Universal Robots PolyScope program: shaft_v1.urp

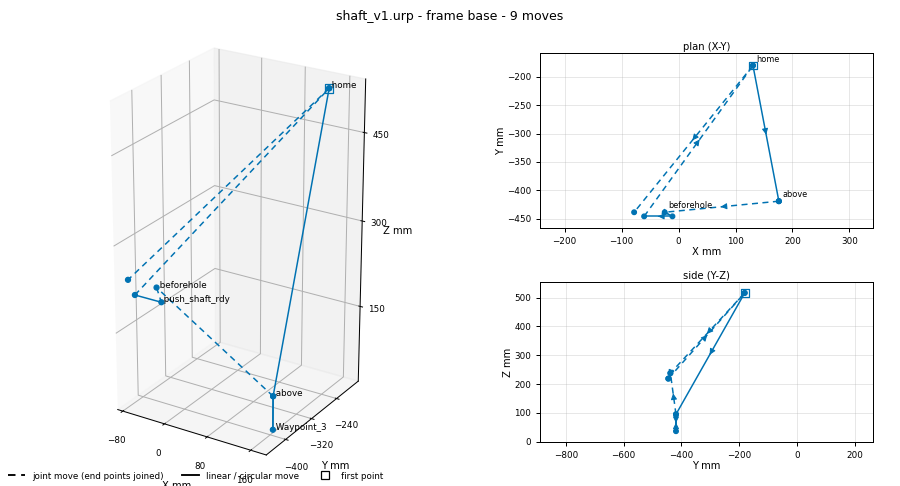
[picture p0: tool path of shaft_v1.urp in frame base, 9 of 9 moves have a stored position in this frame; points joined in program order, loops and branches not executed]
Program shaft_v1 (installation=default directory=/programs/wrs2020 createdIn=5.7.0.90932 lastSavedIn=5.7.0.90932 robotSerialNumber=20205500607)
Calibrated DH parameters: a=[0.000096, -0.337, -0.383372, 0.000118, 0.000015, 0]; d=[0.162724, 79.377998, -95.545185, 16.300583, 0.099689, 0.099499]; alpha=[1.569249, 0.003272, 0.005201, 1.570041, -1.570219, 0]; deltaTheta=[0, 0.65664, 5.410619, 0.215927, -0.000001, 0]
Robot Program (runOnlyOnce=true)
  MoveJ speed 180 deg/s, acceleration 80 deg/s^2 (useActiveTCP=true) feature=Base
    Waypoint home: TCP in base x=130.635 y=-180.692 z=515.97 mm, rx=-0.0117 ry=-3.1402 rz=-0.0315 rad; joints [89.951, -120.324, 80.212, -48.705, -89.957, -0.002] deg; TCP offset x=0 y=0 z=165 mm, rx=0 ry=0 rz=0 rad
  URCap Gripper (Robotiq_Grippers, Robotiq Inc.) dataModel(position=40.0, force=100.0, speed=100.0, positionInDouble=40.0, forceInDouble=100.0, speedInDouble=100.0, slaveIds=[9], blocking=true)
  MoveL speed 250 mm/s, acceleration 1200 mm/s^2 (useActiveTCP=true) feature=Base
    Waypoint above: TCP in base x=176.103 y=-418.817 z=95.382 mm, rx=2.2322 ry=2.1885 rz=0.0336 rad; joints [94.991, -88.211, 123.574, -125.231, -88.184, 96.136] deg
    Waypoint Waypoint_3: TCP in base x=176.103 y=-418.817 z=36.839 mm, rx=2.2322 ry=2.1885 rz=0.0336 rad; joints [94.966, -81.879, 127.739, -135.729, -88.195, 96.172] deg
  URCap Gripper (Robotiq_Grippers, Robotiq Inc.) dataModel(position=100.0, force=100.0, speed=100.0, positionInDouble=100.0, forceInDouble=100.0, speedInDouble=100.0, slaveIds=[9], blocking=true)
  MoveL speed 250 mm/s, acceleration 1200 mm/s^2 (useActiveTCP=true) feature=Base
    Waypoint above: TCP in base x=176.103 y=-418.817 z=95.382 mm, rx=2.2322 ry=2.1885 rz=0.0336 rad; joints [94.991, -88.211, 123.574, -125.231, -88.184, 96.136] deg
  MoveJ speed 60 deg/s, acceleration 80 deg/s^2 (useActiveTCP=true) feature=Base
    Waypoint beforehole: TCP in base x=-24.236 y=-438.216 z=237.961 mm, rx=2.1821 ry=2.2311 rz=0.0137 rad; joints [68.566, -99.136, 110.829, -101.657, -88.409, 67.166] deg
  MoveL speed 20 mm/s, acceleration 500 mm/s^2 (useActiveTCP=true) feature=Base
    SuppressedNode
      Waypoint athole: TCP in base x=-43.043 y=-438.482 z=237.002 mm, rx=2.1821 ry=2.2311 rz=0.0137 rad; joints [66.199, -98.823, 110.698, -101.787, -88.409, 64.799] deg
    MoveDirectionNode (selectedDirection=YMinus) feature=Joint_6_name
      Until TOOL_CONTACT_DETECTION (allowActions=false retraction=0 decelerationAcceleration=3 decelerationAngularAcceleration=34.906585)
  MoveL speed 250 mm/s, acceleration 1200 mm/s^2 (useActiveTCP=true) feature=Base
    MoveDirectionNode (selectedDirection=ZPlus)
      Until DISTANCE (allowActions=false deceleration=3 distanceNodeType=STOP) Distance=0.002; motionParameters(blendRadius=0)
  Force Frame feature=Joint_6_name; selection=[0, 1, 0, 0, 0, 0]; wrench=[-20, -20, 0, 0, 0, 0]; limitsForce=[0.01, 0.01, 0.005, 1.047198, 1.047198, 1.047198]; limitsMotion=[0.1, 0.1, 0.1, 0.349066, 0.349066, 0.349066]
    Wait Sleep waitTime=3
    SuppressedNode
      Loop Counting (count=10) loopVariable(name=Loop_2)
        Force Frame feature=Base; selection=[1, 0, 1, 0, 0, 0]; wrench=[-10, 5, 5, 0, 0, 0]; limitsForce=[0.01, 0.01, 0.01, 1.047198, 1.047198, 1.047198]; limitsMotion=[0.1, 0.1, 0.1, 0.349066, 0.349066, 0.349066]
          Wait Sleep waitTime=2
        Force Frame feature=Base; selection=[1, 0, 1, 0, 0, 0]; wrench=[-10, 5, -5, 0, 0, 0]; limitsForce=[0.01, 0.01, 0.01, 1.047198, 1.047198, 1.047198]; limitsMotion=[0.1, 0.1, 0.1, 0.349066, 0.349066, 0.349066]
          Wait Sleep waitTime=2
        Force Frame feature=Base; selection=[1, 1, 0, 0, 0, 0]; wrench=[-10, 5, 5, 0, 0, 0]; limitsForce=[0.01, 0.01, 0.01, 1.047198, 1.047198, 1.047198]; limitsMotion=[0.1, 0.1, 0.1, 0.349066, 0.349066, 0.349066]
          Wait Sleep waitTime=2
        Force Frame feature=Base; selection=[1, 1, 0, 0, 0, 0]; wrench=[-10, -5, 5, 0, 0, 0]; limitsForce=[0.01, 0.01, 0.01, 1.047198, 1.047198, 1.047198]; limitsMotion=[0.1, 0.1, 0.1, 0.349066, 0.349066, 0.349066]
          Wait Sleep waitTime=2
    'spiral motion'
    SuppressedNode
      Loop Counting (count=30) loopVariable(name=Loop_1)
        MoveL speed 250 mm/s, acceleration 1200 mm/s^2 (useActiveTCP=true) feature=Base
          MoveDirectionNode (toolParams=0.005, 0.02) expression=[sin((Loop_1-1)/6*3.141),0.0,-cos((Loop_1-1)/6*3.141)]; feature=Joint_6_name
            Until DISTANCE (allowActions=false deceleration=3 distanceNodeType=STOP) Distance=0.001; motionParameters(blendRadius=0)
    'grid motion'
    var_1 := 1
    Loop While (checkContinuously=true) expression=( pose_dist(get_actual_tcp_pose(), fully_inserted) > 0.005) and  (var_1 < 6)
      MoveL speed 250 mm/s, acceleration 1200 mm/s^2 (useActiveTCP=true) feature=Base
        MoveDirectionNode (selectedDirection=XPlus toolParams=0.005, 0.02) feature=Joint_6_name
          Until DISTANCE (allowActions=false deceleration=3 distanceNodeType=STOP) Distance=0.0005; motionParameters(blendRadius=0)
        MoveDirectionNode (selectedDirection=ZMinus toolParams=0.005, 0.02) feature=Joint_6_name
          Until DISTANCE (allowActions=false deceleration=3 distanceNodeType=STOP) Distance=0.0005; motionParameters(blendRadius=0)
        MoveDirectionNode (selectedDirection=XMinus toolParams=0.005, 0.02) feature=Joint_6_name
          Until DISTANCE (allowActions=false deceleration=3 distanceNodeType=STOP) Distance=0.0005; motionParameters(blendRadius=0)
        MoveDirectionNode (selectedDirection=XMinus toolParams=0.005, 0.02) feature=Joint_6_name
          Until DISTANCE (allowActions=false deceleration=3 distanceNodeType=STOP) Distance=0.0005; motionParameters(blendRadius=0)
        MoveDirectionNode (selectedDirection=ZPlus toolParams=0.005, 0.02) feature=Joint_6_name
          Until DISTANCE (allowActions=false deceleration=3 distanceNodeType=STOP) Distance=0.0005; motionParameters(blendRadius=0)
        MoveDirectionNode (selectedDirection=XPlus toolParams=0.005, 0.02) feature=Joint_6_name
          Until DISTANCE (allowActions=false deceleration=3 distanceNodeType=STOP) Distance=0.0005; motionParameters(blendRadius=0)
        MoveDirectionNode (selectedDirection=XPlus toolParams=0.005, 0.02) feature=Joint_6_name
          Until DISTANCE (allowActions=false deceleration=3 distanceNodeType=STOP) Distance=0.0005; motionParameters(blendRadius=0)
        MoveDirectionNode (selectedDirection=ZPlus toolParams=0.005, 0.02) feature=Joint_6_name
          Until DISTANCE (allowActions=false deceleration=3 distanceNodeType=STOP) Distance=0.0005; motionParameters(blendRadius=0)
        MoveDirectionNode (selectedDirection=XMinus toolParams=0.005, 0.02) feature=Joint_6_name
          Until DISTANCE (allowActions=false deceleration=3 distanceNodeType=STOP) Distance=0.0005; motionParameters(blendRadius=0)
        MoveDirectionNode (selectedDirection=XMinus toolParams=0.005, 0.02) feature=Joint_6_name
          Until DISTANCE (allowActions=false deceleration=3 distanceNodeType=STOP) Distance=0.0005; motionParameters(blendRadius=0)
        MoveDirectionNode (selectedDirection=ZMinus toolParams=0.005, 0.02) feature=Joint_6_name
          Until DISTANCE (allowActions=false deceleration=3 distanceNodeType=STOP) Distance=0.0005; motionParameters(blendRadius=0)
        MoveDirectionNode (selectedDirection=XPlus toolParams=0.005, 0.02) feature=Joint_6_name
          Until DISTANCE (allowActions=false deceleration=3 distanceNodeType=STOP) Distance=0.0005; motionParameters(blendRadius=0)
      MoveL speed 250 mm/s, acceleration 1200 mm/s^2 (useActiveTCP=true) feature=Base
        MoveDirectionNode (selectedDirection=XPlus toolParams=0.005, 0.02) feature=Joint_6_name
          Until DISTANCE (allowActions=false deceleration=3 distanceNodeType=STOP) Distance=0.001; motionParameters(blendRadius=0)
        MoveDirectionNode (selectedDirection=ZMinus toolParams=0.005, 0.02) feature=Joint_6_name
          Until DISTANCE (allowActions=false deceleration=3 distanceNodeType=STOP) Distance=0.001; motionParameters(blendRadius=0)
        MoveDirectionNode (selectedDirection=XMinus toolParams=0.005, 0.02) feature=Joint_6_name
          Until DISTANCE (allowActions=false deceleration=3 distanceNodeType=STOP) Distance=0.001; motionParameters(blendRadius=0)
        MoveDirectionNode (selectedDirection=XMinus toolParams=0.005, 0.02) feature=Joint_6_name
          Until DISTANCE (allowActions=false deceleration=3 distanceNodeType=STOP) Distance=0.001; motionParameters(blendRadius=0)
        MoveDirectionNode (selectedDirection=ZPlus toolParams=0.005, 0.02) feature=Joint_6_name
          Until DISTANCE (allowActions=false deceleration=3 distanceNodeType=STOP) Distance=0.001; motionParameters(blendRadius=0)
        MoveDirectionNode (selectedDirection=XPlus toolParams=0.005, 0.02) feature=Joint_6_name
          Until DISTANCE (allowActions=false deceleration=3 distanceNodeType=STOP) Distance=0.001; motionParameters(blendRadius=0)
        MoveDirectionNode (selectedDirection=XPlus toolParams=0.005, 0.02) feature=Joint_6_name
          Until DISTANCE (allowActions=false deceleration=3 distanceNodeType=STOP) Distance=0.001; motionParameters(blendRadius=0)
        MoveDirectionNode (selectedDirection=ZPlus toolParams=0.005, 0.02) feature=Joint_6_name
          Until DISTANCE (allowActions=false deceleration=3 distanceNodeType=STOP) Distance=0.001; motionParameters(blendRadius=0)
        MoveDirectionNode (selectedDirection=XMinus toolParams=0.005, 0.02) feature=Joint_6_name
          Until DISTANCE (allowActions=false deceleration=3 distanceNodeType=STOP) Distance=0.001; motionParameters(blendRadius=0)
        MoveDirectionNode (selectedDirection=XMinus toolParams=0.005, 0.02) feature=Joint_6_name
          Until DISTANCE (allowActions=false deceleration=3 distanceNodeType=STOP) Distance=0.001; motionParameters(blendRadius=0)
        MoveDirectionNode (selectedDirection=ZMinus toolParams=0.005, 0.02) feature=Joint_6_name
          Until DISTANCE (allowActions=false deceleration=3 distanceNodeType=STOP) Distance=0.001; motionParameters(blendRadius=0)
        MoveDirectionNode (selectedDirection=XPlus toolParams=0.005, 0.02) feature=Joint_6_name
          Until DISTANCE (allowActions=false deceleration=3 distanceNodeType=STOP) Distance=0.001; motionParameters(blendRadius=0)
      var_1 := var_1+1
  URCap Gripper (Robotiq_Grippers, Robotiq Inc.) dataModel(position=0.0, force=100.0, speed=100.0, positionInDouble=0.0, forceInDouble=100.0, speedInDouble=100.0, slaveIds=[9], blocking=true)
  MoveJ speed 60 deg/s, acceleration 80 deg/s^2 (useActiveTCP=true) feature=Base
    SuppressedNode
      Waypoint ready_to_push: TCP in base x=-56.908 y=-572.13 z=223.439 mm, rx=2.1027 ry=-2.324 rz=0.0706 rad; joints [70.064, -80.555, 94.786, -105.746, -87.55, -104.25] deg
    Waypoint push_shaft_rdy: TCP in base x=-10.71 y=-445.424 z=219.069 mm, rx=2.1821 ry=2.2311 rz=0.0137 rad; joints [70.63, -97.545, 112.338, -104.806, -88.405, 69.25] deg
  SuppressedNode
    URCap Gripper (Robotiq_Grippers, Robotiq Inc.) dataModel(position=52.94117647058823, force=100.0, speed=100.0, positionInDouble=52.94117647058823, forceInDouble=100.0, speedInDouble=100.0, slaveIds=[9], blocking=true)
  URCap Gripper (Robotiq_Grippers, Robotiq Inc.) dataModel(position=100.0, force=100.0, speed=100.0, positionInDouble=100.0, forceInDouble=100.0, speedInDouble=100.0, slaveIds=[9], blocking=true)
  SuppressedNode
    Force Frame feature=Joint_6_name; selection=[0, 1, 0, 0, 0, 0]; wrench=[0, -20, 20, 0, 0, 0]; limitsForce=[0.15, 0.01, 0.01, 1.047198, 1.047198, 1.047198]; limitsMotion=[0.1, 0.1, 0.1, 0.349066, 0.349066, 0.349066]
      Wait Sleep waitTime=20
  MoveL speed 10 mm/s, acceleration 1200 mm/s^2 (useActiveTCP=true) feature=Base
    Waypoint push_shaft: TCP in base x=-60.352 y=-445.424 z=219.069 mm, rx=2.1821 ry=2.2311 rz=0.0137 rad; joints [64.456, -96.881, 111.731, -104.723, -88.406, 63.074] deg
  MoveJ speed 180 deg/s, acceleration 80 deg/s^2 (useActiveTCP=true) feature=Base
    Waypoint home: TCP in base x=130.635 y=-180.692 z=515.97 mm, rx=-0.0117 ry=-3.1402 rz=-0.0315 rad; joints [89.951, -120.324, 80.212, -48.705, -89.957, -0.002] deg
  Halt
  MoveJ speed 60 deg/s, acceleration 80 deg/s^2 (useActiveTCP=true) feature=Base
    Waypoint fully_inserted referenceName=fully_inserted: TCP in base x=-77.923 y=-438.216 z=237.961 mm, rx=2.1821 ry=2.2311 rz=0.0137 rad; joints [61.917, -98.126, 109.947, -101.635, -88.415, 60.516] deg
